Staubli VAL3: start.pgx

program start()
begin
  // Se pone en marcha la aplicacion

  // Se inicializar la aplicacion
  call inicializar()

  taskCreate "Pirámide",100,Piramide()
  taskCreate "mcp",100,mcp()
end
